Staubli VAL3: showTrsf.pgx

program showTrsf(trsf x_tTrsf, string& x_sTrsf[])
begin
  x_sTrsf="("+toString("",x_tTrsf.x)+","+toString("",x_tTrsf.y)+","+toString("",x_tTrsf.z)+","+toString("",x_tTrsf.rx)+","+toString("",x_tTrsf.ry)+","+toString("",x_tTrsf.rz)+")"
end
